PROGRAM MAIN
VAR
	MachineControl : ControlPanel;
	MachineLamps : LampControl := (Controller := MachineControl);
END_VAR

MachineLamps.Cycle();

END_PROGRAM

(* stored: Version 1.1.0.1, ProductVersion 3.1.4024.12
   POU MAIN: Id {cfeb14e3-e49d-4d05-801a-00ad13175c31}, SpecialFunc None *)
